{attribute 'GeneratedUsingTerminal: EP5101-0002-0016'}
{attribute addProperty BoxType "EP5101-0002-0016"}
{attribute addProperty Id "ENC_Status_compactAT %I*ENC_Status_compact_F4F8958316ENC_Control_compactAT %Q*ENC_Control_compact_E6DC9B254WcStateAT %I*WcState_9091E0EB2InfoDataAT %I*InfoData_32EB74EA10"}
{attribute addProperty CRC "2276227279"}
{attribute addProperty Size "32"}
TYPE EP5101_87AC78CF :
STRUCT
	{attribute addProperty Name "ENC_Status_compact"}
	ENC_Status_compact : ENC_Status_compact_F4F89583;
	{attribute addProperty Name "ENC_Control_compact"}
	ENC_Control_compact : ENC_Control_compact_E6DC9B25;
	{attribute addProperty Name "WcState"}
	WcState : WcState_9091E0EB;
	{attribute addProperty Name "InfoData"}
	InfoData : InfoData_32EB74EA;
END_STRUCT
END_TYPE

(* stored: Version 1.2.0.0, ProductVersion 3.1.4024.9
   DUT EP5101_87AC78CF: Id {bce20810-55f3-418c-8279-3a144b36437c} *)
